{attribute 'Tc2GvlVarNames'}
VAR_GLOBAL
	IN_Stromzaehler AT %I* 	: ST_KL6781inData22B;
	OUT_Stromzaehler AT %Q* : ST_KL6781outData22B;
	IN_WZaehler AT %I* 	: ST_KL6781inData22B;
	OUT_WZaehler AT %Q* : ST_KL6781outData22B;
	IN_WZaehler2 AT %I* 	: ST_KL6781inData22B;
	OUT_WZaehler2 AT %Q* : ST_KL6781outData22B;
	IN_WZaehler_Basement AT %I* 	: ST_KL6781inData22B;
	OUT_WZaehler_Basement AT %Q* : ST_KL6781outData22B;
	
	(*
			[1] ETA_3111U1006XHE321XXXXXXZ01, ELT_Zaehler_BHKW_321_01
			Primaer-Adresse = 1
			Seriennummer = 3999427
			[2] ETA_3111U1006XHE322XXXXXXZ01, ELT_Zaehler_BHKW_322_01
			Primaer-Adresse = 2
			Seriennummer = 3999432
			[3] ETA_3111U1006BEST001XXXXXXZ01, ELT_Zaehler_Buerotrakt_01
			Primaer-Adresse = 3
			Seriennummer = 120267
			[4] ETA_3111U1006BEST002XXXXXXZ01, ELT_Zaehler_Gebaede_01
			Primaer-Adresse = 4
			Seriennummer = 205684
			[5] ETA_3111U1006BEST003XXXXXXZ01, ELT_Zaehler_Halle_TGA_01
			Primaer-Adresse = 5
			Seriennummer = 120264
			[6] ETA_3111EG005BEST004XXXXXXZ01, ELT_Zaehler_Halle_Licht_01
			Primaer-Adresse = 6
			Seriennummer = 214516
			[7] ETA_3111U1006BEST007XXXXXXZ01, GAS_Zaehler BHKW_007_01
			Primaer-Adresse = 7
			Seriennummer = 42078747
			[8] ETA_3111U1006BEST008XXXXXXZ01, GAS_Zaehler BHKW_008_01
			Primaer-Adresse = 8
			Seriennummer = 42078748
			[9] ETA_3111U1006BEST071XXXXXXZ01, WAERME_Zaehler WP_945_4371_01
			Primaer-Adresse = 71
			Seriennummer = 67694371
			[10] ETA_3111U1006BEST072XXXXXXZ01, WAERME_Zaehler WP_945_4372_01
			Primaer-Adresse = 72
			Seriennummer = 67694372
	*)
	Kommunikation_MBus	: ST_MBUS_Communication;
	Komm_MBus_WZaehler	: ST_MBUS_Communication;
	Komm_MBus_WZaehler2	: ST_MBUS_Communication;
	Komm_MBus_WZaehler_Basement	: ST_MBUS_Communication;

	aTelegramm_WMZ350 						: ARRAY[1..cMBUS_MaxTelegrams] OF ST_MBus_Data2;
	aTelegramm_WMZ305 						: ARRAY[1..cMBUS_MaxTelegrams] OF ST_MBus_Data2;
	aTelegramm_WMZ100 						: ARRAY[1..cMBUS_MaxTelegrams] OF ST_MBus_Data2;
	aTelegramm_WMZ300 						: ARRAY[1..cMBUS_MaxTelegrams] OF ST_MBus_Data2;
	aTelegramm_WMZ245 						: ARRAY[1..cMBUS_MaxTelegrams] OF ST_MBus_Data2;
	aTelegramm_WMZ235 						: ARRAY[1..cMBUS_MaxTelegrams] OF ST_MBus_Data2;
	aTelegramm_WMZ405 						: ARRAY[1..cMBUS_MaxTelegrams] OF ST_MBus_Data2;
	aTelegramm_WMZ425 						: ARRAY[1..cMBUS_MaxTelegrams] OF ST_MBus_Data2;
	aTelegramm_WMZ455 						: ARRAY[1..cMBUS_MaxTelegrams] OF ST_MBus_Data2;
	aTelegramm_WMZ342 						: ARRAY[1..cMBUS_MaxTelegrams] OF ST_MBus_Data2;
	
	
	aTelegramm_WMZ900 						: ARRAY[1..cMBUS_MaxTelegrams] OF ST_MBus_Data2;
	aTelegramm_WMZ935 						: ARRAY[1..cMBUS_MaxTelegrams] OF ST_MBus_Data2;
	
	aTelegramm_WMZ135						: ARRAY[1..cMBUS_MaxTelegrams] OF ST_MBus_Data2;
	aTelegramm_WMZ138						: ARRAY[1..cMBUS_MaxTelegrams] OF ST_MBus_Data2;
	aTelegramm_WMZ105						: ARRAY[1..cMBUS_MaxTelegrams] OF ST_MBus_Data2;
	aTelegramm_WMZ710						: ARRAY[1..cMBUS_MaxTelegrams] OF ST_MBus_Data2;
	aTelegramm_WMZ205						: ARRAY[1..cMBUS_MaxTelegrams] OF ST_MBus_Data2;
	aTelegramm_WMZ720						: ARRAY[1..cMBUS_MaxTelegrams] OF ST_MBus_Data2;
	
	Telegramm_WZ_Brennwerttherme			: ARRAY[1..cMBUS_MaxTelegrams] OF ST_MBus_Data2;
	Telegramm_WZ_BHKW_1						: ARRAY[1..cMBUS_MaxTelegrams] OF ST_MBus_Data2;
	Telegramm_WZ_BHKW_2						: ARRAY[1..cMBUS_MaxTelegrams] OF ST_MBus_Data2;
	Telegramm_WZ_Druckluftkompressor		: ARRAY[1..cMBUS_MaxTelegrams] OF ST_MBus_Data2;
	Telegramm_WZ_PWT_1						: ARRAY[1..cMBUS_MaxTelegrams] OF ST_MBus_Data2;
	Telegramm_WZ_Ofenkuehlung				: ARRAY[1..cMBUS_MaxTelegrams] OF ST_MBus_Data2;
	Telegramm_WZ_Abwaerme_Ofen_Abgasfackel	: ARRAY[1..cMBUS_MaxTelegrams] OF ST_MBus_Data2;


	Telegramm_SZ_BHKW_321		: ARRAY[1..cMBUS_MaxTelegrams] OF ST_MBus_Data2;
	Telegramm_SZ_BHKW_322		: ARRAY[1..cMBUS_MaxTelegrams] OF ST_MBus_Data2;
	Telegramm_SZ_Buerotrakt		: ARRAY[1..cMBUS_MaxTelegrams] OF ST_MBus_Data2;
	Telegramm_SZ_Gebaeude		: ARRAY[1..cMBUS_MaxTelegrams] OF ST_MBus_Data2;
	Telegramm_SZ_Halle_TGA		: ARRAY[1..cMBUS_MaxTelegrams] OF ST_MBus_Data2;
	Telegramm_SZ_Halle_Licht	: ARRAY[1..cMBUS_MaxTelegrams] OF ST_MBus_Data2;

	Telegramm_GZ_BHKW_321		: ARRAY[1..cMBUS_MaxTelegrams] OF ST_MBus_Data2;
	Telegramm_GZ_BHKW_322		: ARRAY[1..cMBUS_MaxTelegrams] OF ST_MBus_Data2;

	Telegramm_WZ_4371_WP_946	: ARRAY[1..cMBUS_MaxTelegrams] OF ST_MBus_Data2;
	Telegramm_WZ_4372_WP_946	: ARRAY[1..cMBUS_MaxTelegrams] OF ST_MBus_Data2;
	
	maxNumberOfNodes :INT := 22;
	cMSRLIBMaxNumberOfMBusDevices : BYTE := 18;	(*~
				Maximale Anzahl an MBus Geräten, die von der MSRlib unterstützt werden.
				Diese Konstante wird auch für die DP-Historisierung verwendet und muss grösser 6 (Anzahl der Basisdatentypen) sein.
				*)
	cMBUS_MaxData : INT := 40;
	(*cMBUS_MaxTelegrams : INT := 2;
	cMBUS_MaxCom : INT := 1;*)

END_VAR

(* stored: Version 1.1.0.1, ProductVersion 3.1.4024.10
   GVL M_Bus: Id {09f3b77d-e1a8-4a2e-b9d8-80d0df79e368} *)
